// TIA Portal project "counter" (V14)

(* hardware
DEVICE "S7-1200 station_1"  S7-1200 Station
   slot 0: "Rack_0"  S7-1200 Rack  Rack  V1.0
   slot 1: "PLC_1"  CPU 1212C DC/DC/DC  6ES7 212-1AE40-0XB0  V4.2
DEVICE "HMI_1"  KTP400 Basic PN
   slot 0: "KTP400 Basic PN"  KTP400 Basic PN  6AV2 123-2DB03-0AX0  14.0.1.0
   slot 1: "HMI_RT_1"  KTP400 Basic PN  6AV2 123-2DB03-0AX0  14.0.1.0
   slot 5: "HMI_1.IE_CP_1"  PROFINET Interface  14.0.1.0
      slot 1: "PROFINET Interface_1"  PROFINET Interface
         slot 1: "Port_1"  Port
*)

// ===== PLC "PLC_1"  CPU 1212C DC/DC/DC =====

VAR_GLOBAL   // PLC tag table "Default tag table"
   "Tag_1" AT %I0.3 : Bool;
   "Tag_2" AT %I0.1 : Bool;
   "Tag_3" AT %Q0.3 : Bool;
   "Tag_4" AT %Q0.0 : Bool;
   "Tag_5" AT %Q0.2 : Bool;
   "Tag_6" AT %I0.0 : Bool;
   "Tag_7" AT %M0.0 : Bool;
   "Tag_8" AT %I0.2 : Bool;
   "Tag_9" AT %M0.2 : Bool;
   "START_HMI" AT %M0.1 : Bool;
   "STOP_HMI" AT %M0.3 : Bool;
   "HIEN THI 1" AT %MW2 : Int;
   "RESET_HMI1" AT %M0.4 : Bool;
   "HIEN THI 2" AT %MD4 : Time;
   "HIEN THI 3" AT %MD8 : Time;
   "HIEN THI 4" AT %MW12 : Int;
END_VAR

// folder: System blocks/Program resources

DATA_BLOCK "IEC_Counter_0_DB"   // DB2
{ S7_Optimized_Access := 'TRUE' }
AUTHOR : Simatic
FAMILY : IEC
NAME : CNTR
VERSION : 1.0
// stored: InstanceOfName IEC_COUNTER
"IEC_COUNTER"
BEGIN
END_DATA_BLOCK

DATA_BLOCK "t1"   // DB3
{ S7_Optimized_Access := 'TRUE' }
AUTHOR : Simatic
FAMILY : IEC
NAME : IEC_TMR
VERSION : 1.0
// stored: InstanceOfName IEC_TIMER
"IEC_TIMER"
BEGIN
END_DATA_BLOCK

// folder: (top level)

ORGANIZATION_BLOCK "Main"   // OB1, LAD, ProgramCycle
TITLE = "Main Program Sweep (Cycle)"
{ S7_Optimized_Access := 'TRUE' }
VERSION : 0.1
   VAR_INPUT
      Initial_Call : Bool;   // Initial call of this OB
      Remanence : Bool;   // =True, if remanent data are available
   END_VAR
   VAR_TEMP
      RESET_HMI : Bool;
   END_VAR
   VAR_TEMP   // added for the SCL form of the ladder/FBD networks
      _w1 : Bool;
   END_VAR
BEGIN

REGION Network 1
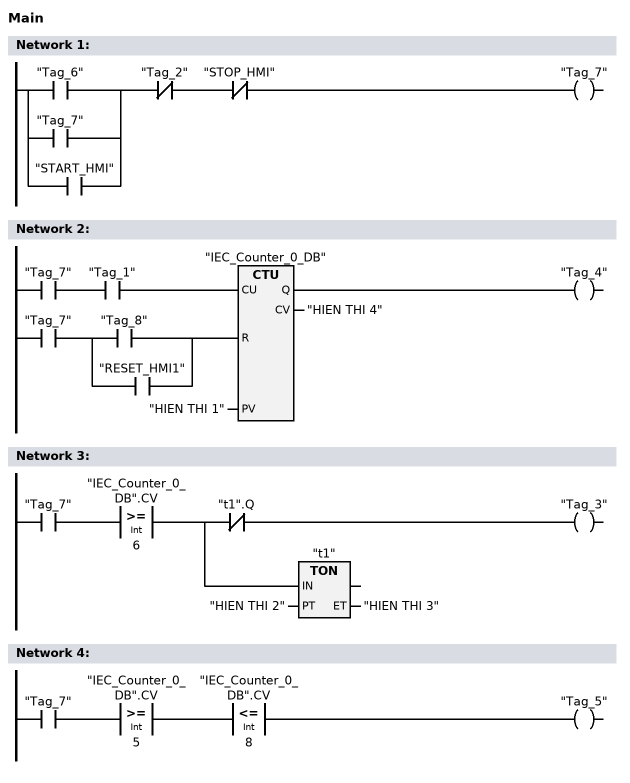
   RUNG wire#powerrail
      Contact( "Tag_6" )
      wire#w1
      I_Contact( "Tag_2" )
      I_Contact( "STOP_HMI" )
      Coil( "Tag_7" )
   END_RUNG
   RUNG wire#powerrail
      Contact( "Tag_7" )
   END_RUNG wire#w1
   RUNG wire#powerrail
      Contact( "START_HMI" )
   END_RUNG wire#w1
   // the same network as SCL:
   "Tag_7" := ("Tag_6" OR "Tag_7" OR "START_HMI") AND NOT "Tag_2" AND NOT "STOP_HMI";
END_REGION

REGION Network 2
   "IEC_Counter_0_DB".CTU(CU := "Tag_7" AND "Tag_1",
                          R := "Tag_7" AND ("Tag_8" OR "RESET_HMI1"),
                          PV := "HIEN THI 1",
                          CV => "HIEN THI 4");
   "Tag_4" := "IEC_Counter_0_DB".Q;
END_REGION

REGION Network 3
   #_w1 := "Tag_7" AND ("IEC_Counter_0_DB".CV >= 6);
   "Tag_3" := #_w1 AND NOT "t1".Q;
   "t1".TON(IN := #_w1, PT := "HIEN THI 2", ET => "HIEN THI 3");
END_REGION

REGION Network 4
   RUNG wire#powerrail
      Contact( "Tag_7" )
      { S7_Templates := "SrcType := Int" } GE_Contact(in1 := "IEC_Counter_0_DB".CV, in2 := 5)
      { S7_Templates := "SrcType := Int" } LE_Contact(in1 := "IEC_Counter_0_DB".CV, in2 := 8)
      Coil( "Tag_5" )
   END_RUNG
   // the same network as SCL:
   "Tag_5" := "Tag_7" AND ("IEC_Counter_0_DB".CV >= 5) AND ("IEC_Counter_0_DB".CV <= 8);
END_REGION
END_ORGANIZATION_BLOCK

(* ===== HMI "HMI_RT_1" =====
system functions are stored by id; their names below are inferred from use
connection "HMI_Connection_1": ETHERNET, SMART_S7_1200_OMS

HMI tags "Default tag table"
   "START_HMI" : Bool = PLC START_HMI AT %M0.1, 100 ms
   "STOP_HMI" : Bool = PLC STOP_HMI AT %M0.3, 100 ms
   "RESET_HMI1" : Bool = PLC RESET_HMI1 AT %M0.4, 100 ms
   "Tag_4" : Bool = PLC Tag_4 AT %Q0.0, 100 ms
   "HIEN THI 1" : Int = PLC "HIEN THI 1" AT %MW2, 100 ms
   "HIEN THI 2" : Time = PLC "HIEN THI 2" AT %MD4, 100 ms
   "HIEN THI 3" : Time = PLC "HIEN THI 3" AT %MD8, 100 ms
   "HIEN THI 4" : Int = PLC "HIEN THI 4" AT %MW12, 100 ms

Template "Template_1" 480x272
   Button "Exit" at 388,227 size 63x44; TextOff 'Exit'; PictureOff "ExitRuntime_KTP400_Basic_PN_TR"; PictureOn "ExitRuntime_KTP400_Basic_PN_TR"
      on Release: StopRuntime(0)
   Button "Template_Button" at 268,227 size 63x44; TextOff 'Text'
   Button "Template_Button_1" at 148,227 size 63x44; TextOff 'Text'
   Button "Start screen" at 28,227 size 63x44; TextOff 'Start screen'; PictureOff "NavigateHome_KTP400_Basic_PN_TR"; PictureOn "NavigateHome_KTP400_Basic_PN_TR"
      on Release: ActivateScreen("Root screen", 0)

screen "Root screen" 480x272, template "Template_1"
   TextField "Text field_1" at 108,18 size 265x27; Text 'LAP TRINH HMI PROJECT1'
   Button "Button_1" at 27,153 size 96x32; TextOff 'Start'
      on Press: SetBit("START_HMI")
      on Release: ResetBit("START_HMI")
   Button "Button_2" at 139,153 size 96x32; TextOff 'Stop'
      on Press: SetBit("STOP_HMI")
      on Release: ResetBit("STOP_HMI")
   Button "Button_3" at 254,153 size 96x32; TextOff 'Reset'
      on Press: SetBit("RESET_HMI1")
      on Release: ResetBit("RESET_HMI1")
   Circle "Circle_1" at 403,153 size 48x48
      Appearance <- "Tag_4"
   IOField "I/O field_1" at 22,98 size 96x32; FormatPattern s99999
      ProcessValue <- "HIEN THI 1"
   IOField "I/O field_2" at 254,99 size 96x32; FormatPattern s9999999999
      ProcessValue <- "HIEN THI 2"
   IOField "I/O field_3" at 379,98 size 96x32; FormatPattern s9999999999
      ProcessValue <- "HIEN THI 3"
   IOField "I/O field_4" at 135,99 size 96x32; FormatPattern s99999
      ProcessValue <- "HIEN THI 4"
*)